(* CoDeSys 2.3 export: SENSOR_CAP.EXP *)

(* Data type *)
TYPE Sensor_Cap :
STRUCT
	Activo : BOOL;
END_STRUCT
END_TYPE
